(*

.. <legal notes>

legal notes
=================
| SPDX-FileCopyrightText: © 2025 Oleksandr Tiutyk <trofimich@gmail.com>
| SPDX-License-Identifier: LGPL-3.0-only
| For details check: LGPL-3.0-only_

.. _LGPL-3.0-only: https://www.gnu.org/licenses/lgpl-3.0.en.html

.. </legal notes>

*)

INTERFACE IAbortableProcess EXTENDS IProcess

{attribute 'monitoring' := 'call'}
{attribute 'OPC.UA.DA.Property' := '1'}
{attribute 'OPC.UA.DA.Access' := '1'}
PROPERTY Aborted : BOOL
GET
END_GET
END_PROPERTY

{attribute 'monitoring' := 'call'}
{attribute 'OPC.UA.DA.Property' := '1'}
{attribute 'OPC.UA.DA.Access' := '1'}
PROPERTY Aborting : BOOL
GET
END_GET
END_PROPERTY

{attribute 'monitoring' := 'call'}
{attribute 'OPC.UA.DA.Property' := '1'}
{attribute 'OPC.UA.DA.Access' := '1'}
PROPERTY AbortReason : REFERENCE TO ERROR_MESSAGE
GET
END_GET
END_PROPERTY

{attribute 'monitoring' := 'call'}
{attribute 'OPC.UA.DA.Property' := '1'}
{attribute 'OPC.UA.DA.Access' := '1'}
PROPERTY Busy : BOOL
GET
END_GET
END_PROPERTY

METHOD StartAbort
VAR_INPUT 
	reason : ERROR_MESSAGE := "";
END_VAR
END_METHOD

END_INTERFACE

(* stored: Version 1.1.0.1
   Itf IAbortableProcess: Id {673acb26-d0c2-4ba2-81ae-6136dc542627}
   Property Aborted: Id {1b200195-722a-477c-8d67-52804e0bbba2}
   Get Get: Id {2472e367-f7fc-46ae-95ec-96cab3351e7b}
   Property Aborting: Id {e180feda-a63d-49c7-a58c-a16b8d3b8f36}
   Get Get: Id {8a8427f9-bdb9-4110-be31-f735ab18592d}
   Property AbortReason: Id {14a1cb54-5441-457c-bea8-c28e366481bc}
   Get Get: Id {de5e06a5-9fa3-434b-ba32-89384ee72df0}
   Property Busy: Id {1dc419c8-743c-497e-a28d-604a4ef22e1c}
   Get Get: Id {05d3eb4b-b335-466c-af3e-46b36e8b2e1a}
   Method StartAbort: Id {8c3c78ee-be09-40e9-9b9f-fa08ff8e2858} *)
